FUNCTION_BLOCK AX_FB_R_IO (* Realizes a monostable reset-dominat (with Adapter) *)
  (* Standard: 61499-1; Description: Copyright (c) 2023 Martin Erich Jobst, HR Agrartechnik GmbH This program and the accompanying materials are made available under the terms of the Eclipse Public License 2.0 which is available at https://www.eclipse.org/legal/epl-2.0/ SPDX-License-Identifier: EPL-2.0 *)
  (* Version 3.0, 2025-04-14, Patrick Aigner, changed package *)
  (* Version 1.0, 2023-04-28, Martin Jobst, initial API and implementation and/or initial documentation *)
  PACKAGE adapter::monostableElements;
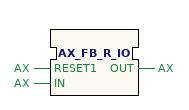
  SOCKETS
    RESET1 : adapter::types::unidirectional::AX; (* Reset *)
    IN : adapter::types::unidirectional::AX; (* Input *)
  END_SOCKETS
  PLUGS
    OUT : adapter::types::unidirectional::AX; (* Output *)
  END_PLUGS
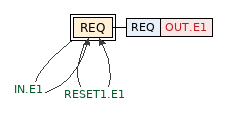
  EC_STATES
    REQ : REQ -> OUT.E1;
  END_STATES
  EC_TRANSITIONS
    REQ TO REQ := RESET1.E1;
    REQ TO REQ := IN.E1;
  END_TRANSITIONS
  ALGORITHM REQ IN ST: (* This algorithm passes the input signal (IN.D1) directly to the output (OUT.D1) during normal operation. However, if the prioritized reset signal (RESET1.D1) is active, it overrides the input and forces the output to FALSE. *)
IF RESET1.D1 THEN
	OUT.D1 := BOOL#FALSE;
ELSE
	OUT.D1 := IN.D1;
END_IF;
  END_ALGORITHM
END_FUNCTION_BLOCK
